Staubli VAL3: motionProgress.pgx

public program motionProgress(num x_nMoveId, num x_nMotProg)
begin

  // display nMoveId and nMotionProgress

  gotoxy(scMonitor, 0,7)
  put(scMonitor, "moveId:")
  gotoxy(scMonitor, 8,7)
  put(scMonitor, x_nMoveId)
  gotoxy(scMonitor, 13,7)
  put(scMonitor, "progress:")
  gotoxy(scMonitor, 23,7)
  put(scMonitor, x_nMotProg)

end
